TEXTLIST TextListSpitUnitState
  0 = 'off'
  1 = 'initializing'
  2 = 'homing'
  3 = 'ready'
  4 = 'moving'
  100 = 'error'
   = ''
END_TEXTLIST

(* stored: Version 1.1.0.1, ProductVersion 3.1.4024.11
   TextList TextListSpitUnitState: Id {d5ea6483-365d-4332-8cd9-83338d1aaa9c} *)
